% RSLogix 500 project TASSSSSS_ED_BAK009.RSS, saved by version 8.10.00.18 %
PROJECT "UNTITLED"    % processor: MicroLogix 1200 %

PROGRAM FILES
  LAD 2   5 rungs

DATA FILES
  O0 OUTPUT  4 elements
  I1 INPUT  4 elements
  S2 STATUS  66 elements
  B3 BINARY  1 elements
  T4 TIMER  1 elements
  C5 COUNTER  2 elements
  R6 CONTROL  1 elements
  N7 INTEGER  1 elements

LADDER 2
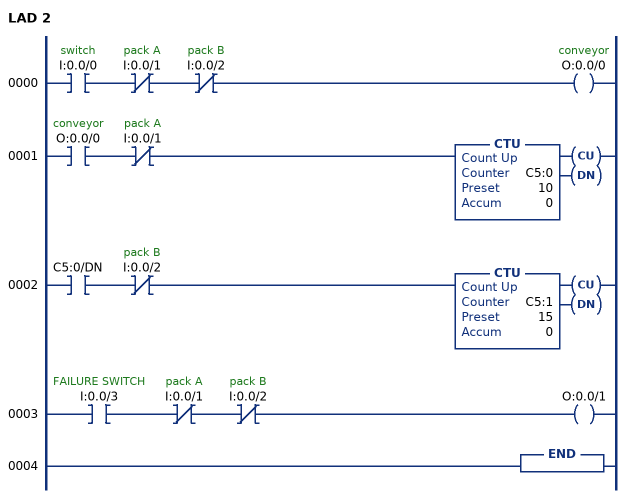
% Rung: 0 %
SOR XIC I:0.0/0 XIO I:0.0/1 XIO I:0.0/2 OTE O:0.0/0 EOR
%   I:0.0/0  "switch" %
%   I:0.0/1  "pack A" %
%   I:0.0/2  "pack B" %
%   O:0.0/0  "conveyor" %
% Rung: 1 %
SOR XIC O:0.0/0 XIO I:0.0/1 CTU C5:0 10 0 EOR
%   O:0.0/0  "conveyor" %
%   I:0.0/1  "pack A" %
% Rung: 2 %
SOR XIC C5:0/DN XIO I:0.0/2 CTU C5:1 15 0 EOR
%   I:0.0/2  "pack B" %
% Rung: 3 %
SOR XIC I:0.0/3 XIO I:0.0/1 XIO I:0.0/2 OTE O:0.0/1 EOR
%   I:0.0/3  "FAILURE SWITCH" %
%   I:0.0/1  "pack A" %
%   I:0.0/2  "pack B" %
% Rung: 4 %
SOR END EOR

DATA TABLE (non-zero values as saved)
DATA C5
% .PRE .ACC %
% C5:0 % 10 0
% C5:1 % 15 0
